FUNCTION_BLOCK InductiveSensor IMPLEMENTS ITF_BinarySensor
VAR_INPUT
END_VAR
VAR_OUTPUT
END_VAR
VAR
	//Hardware
	//{attribute 'OPC.UA.DA' := '1'}
	DI_WPMetallic AT %I* : BOOL;
END_VAR

PROPERTY Value : BOOL
GET
Value := DI_WPMetallic;
END_GET
END_PROPERTY

END_FUNCTION_BLOCK

(* stored: Version 1.1.0.1, ProductVersion 3.1.4024.9
   POU InductiveSensor: Id {a2f4d302-ddcc-4dee-b36e-b3987e5861b4}, SpecialFunc None
   Property Value: Id {68c6e4c5-5f2c-4f9b-b56b-cb3e1b1ac4da}
   Get Get: Id {070b8c31-94e6-4c88-811e-d84153f953f5} *)
